TYPE ST_QrScanProcessConfig :
STRUCT
    // 扫码相对相机角度的工艺偏移；最终以绝对目标角度执行。
    fOffsetAngle : LREAL;
END_STRUCT
END_TYPE

(* stored: Version 1.1.0.1, ProductVersion 3.1.4026.20
   DUT ST_QrScanProcessConfig: Id {126ba197-7969-4017-9ffa-bb3fabda6d37} *)
